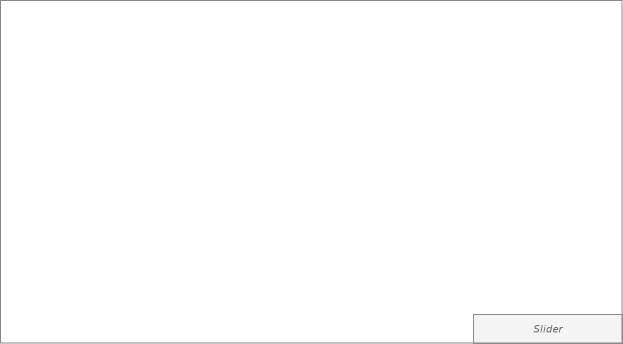
VISUALIZATION Visualization  // 623x344
    Slider (473,314 150x30), variable: MAIN.Ngevraagedwarden, scale 0..100
END_VISUALIZATION

(* stored: Version 1.1.0.1, ProductVersion 3.1.4024.12
   Visu Visualization: Id {9fad7bc7-1754-4c59-906c-75f57efcd747} *)
